(* CoDeSys 2.3 export: EEPROMADRRESS_TS.EXP *)

(* Data type in Diag/Parameter *)
TYPE EEPROMAdrress_ts :
STRUCT
	Page_u8		: USINT;
	IntIndex_u8	: USINT;
END_STRUCT
END_TYPE
